TYPE T_CheckElement :
STRUCT
	eState: E_DecisionState;
	dinActPos_um: DINT;
END_STRUCT
END_TYPE

(* stored: Version 1.1.0.1, ProductVersion 3.1.0.19
   DUT T_CheckElement: Id {97fbcfef-cfc2-43e6-8b57-c9f4e7be8bf7} *)
